// TIA Portal V19 export
DATA_BLOCK "DB_Zwangsziel"   // DB67
{ S7_Optimized_Access := 'FALSE' }
// stored: AutoNumber false
   VAR RETAIN
      Ziel_von_Pos : Array[0..30] of Byte;   // * Feldlänge anpassen
   END_VAR
BEGIN
END_DATA_BLOCK
